// TwinCAT 3 PLC project test_lv2_communication_Http_Rest
// ProgramVersion: 3.1.4020.1
// libraries:
//   Tc2_Standard, * (Beckhoff Automation GmbH)
//   Tc2_System, * (Beckhoff Automation GmbH)
//   Tc3_Module, * (Beckhoff Automation GmbH)
//   tclib_ph_lv2_http, * (Poh)
// project tree:
//   / PlcTask.TcTTO
//   POUs/ MAIN.TcPOU
// (motion and I/O tree: see PLC project ph_lv0)
// real-time tasks:
//   TASK PlcTask: cycle T#10ms, priority 20, ADS port 350

CONFIGURATION test_lv2_communication_Http_Rest
    RESOURCE PLC ON TwinCAT3
        TASK PlcTask(INTERVAL := T#10ms, PRIORITY := 20);
        PROGRAM MAIN WITH PlcTask : MAIN;
    END_RESOURCE
END_CONFIGURATION

// ---- POUs/MAIN.TcPOU
PROGRAM MAIN
VAR
	_VERSION : C_HTTP_VERSION(Major_Version:= 0, Minor_Version:= 0);
	_REQUEST : C_HTTP_REQUEST;
	_REQUEST_PARSE : C_HTTP_REQUEST;
	_RESPONSE : C_HTTP_RESPONSE;
	_RESPONSE_PARSE : C_HTTP_RESPONSE;
	_STRING : STRING(255);
	_STRING_2 : STRING(255);
	_bool1, _bool2, _bool3 : BOOL;
END_VAR

_STRING := _REQUEST.ToString();
_REQUEST_PARSE.Parse('PUT /myUri HTML/1.1$R$NmyHeader: HiHi$R$N$R$NTest this body $R$N');
_STRING_2 := _RESPONSE.ToString();
_RESPONSE_PARSE.Parse('HTML/1.1 200 OK$R$NmyHeader: HiHi$R$N$R$NTest this body $R$N');

END_PROGRAM
